PROGRAM MAIN
VAR
	TestSuite : TestSuite;
	CalculatorTest : CalculatorTest;
	BrokenCalculatorTest: BrokenCalculatorTest;
END_VAR

TcUnit.RUN();

END_PROGRAM

(* stored: Version 1.1.0.1, ProductVersion 3.1.4024.6
   POU MAIN: Id {fe27a7e1-9005-4eae-9b1e-49589e7748de}, SpecialFunc None *)
